{attribute 'qualified_only'}
{attribute 'strict'}
TYPE E_ToolType :
(
	Undefined := 0,
	None,
	Last,
	Tray
);
END_TYPE

(* stored: Version 1.1.0.1, ProductVersion 3.1.4024.5
   DUT E_ToolType: Id {c22aa7e2-c4cc-49dd-b24d-9a7b5388661b} *)
